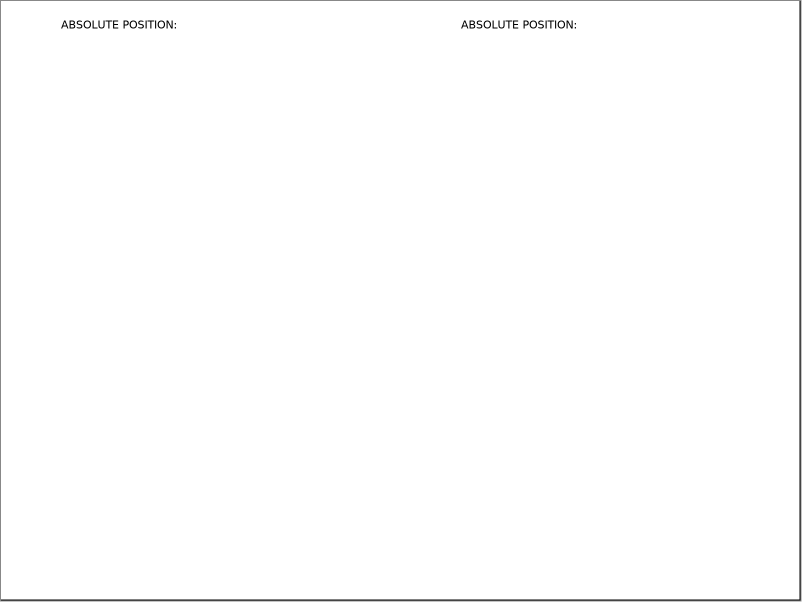
VISUALIZATION F54_Cam_Scaling_V2  // 802x602
    Rectangle (0,0 800x600)
    Label (10,10 170x30), "ABSOLUTE POSITION:"
    Label (410,10 170x30), "ABSOLUTE POSITION:"
END_VISUALIZATION

(* stored: Version 1.1.0.1, ProductVersion 3.1.4022.7
   Visu F54_Cam_Scaling_V2: Id {dd80613f-311b-4e7a-926b-56b29af18c3a} *)
